(* PLC project multi-phase-flow-facility, Generated TextualNotationConverter 1.0 *)
(* stored: creationDateTime 2025-07-30T12:00:00, modificationDateTime 2025-01-30T12:00:00 *)

FUNCTION_BLOCK ANALOG_IN
  VAR_INPUT
    Name : STRING;
    Description : STRING;
    Raw_Signal : REAL;
    PV_High : REAL;
    PV_Low : REAL;
    Scaling_Slope : REAL;
    Scaling_Offset : REAL;
    Alarm_Enable : BOOL;
  END_VAR
  VAR_OUTPUT
    PV : REAL;
    High_Alarm : BOOL;
    Low_Alarm : BOOL;
    General_Fault : BOOL;
  END_VAR

            
          
END_FUNCTION_BLOCK

FUNCTION_BLOCK PID_BASIC
  VAR_INPUT
    Name : STRING;
    Description : STRING;
    AUTO : BOOL;
    PV : REAL;
    SP : REAL;
    MV_MIN : REAL;
    MV_MAX : REAL;
    X0 : REAL;
    KP : REAL;
    TR : REAL;
    TD : REAL;
    PV_High : REAL;
    PV_Low : REAL;
    Deviation_Limit : REAL;
    Inhibit : BOOL;
  END_VAR
  VAR_OUTPUT
    PV_High_Alarm : BOOL;
    PV_Low_Alarm : BOOL;
    Deviation_Alarm : BOOL;
    XOUT : REAL;
  END_VAR

            
          
END_FUNCTION_BLOCK

FUNCTION_BLOCK RATIO_CONTROL
  VAR_INPUT
    Name : STRING;
    Description : STRING;
    Auto : BOOL;
    PrimaryPV : REAL;
    SecondaryPV : REAL;
    RatioSP : REAL;
    Bias : REAL;
    TrimKp : REAL;
    TrimTi : STRING;
    MV_MIN : REAL;
    MV_MAX : REAL;
    ManOut : REAL;
    Inhibit : BOOL;
  END_VAR
  VAR_OUTPUT
    SlaveSP : REAL;
    ActiveRatio : REAL;
    RatioErr : REAL;
  END_VAR

            
          
END_FUNCTION_BLOCK

FUNCTION_BLOCK VALVE_ELECTRIC
  VAR_INPUT
    Name : STRING;
    Description : STRING;
    Control_Signal : REAL;
    Manual_Mode : BOOL;
    Manual_Position : REAL;
    Open_Limit : REAL;
    Close_Limit : REAL;
    Timeout : STRING;
    Inhibit : BOOL;
  END_VAR
  VAR_OUTPUT
    Valve_Position : REAL;
    Feedback_Pos : REAL;
    Valve_Moving : BOOL;
    Position_Error : BOOL;
    Alarm : BOOL;
  END_VAR

            
          
END_FUNCTION_BLOCK

PROGRAM Section2
  VAR
    FT404_GasFlow_PV : REAL;
    FT406_LiquidFlow_PV : REAL;
    FFIC402_LiquidFlow_SP : REAL;
    FIC406_MV_ToCV406 : REAL;
    PT403_SeparatorPressure_PV : REAL;
    PT408_AuxPressure_PV : REAL;
    PIC401_MV_ToCV401 : REAL;
  END_VAR
  VAR
    FT-404 : ANALOG_IN;
    FT-406 : ANALOG_IN;
    PT-403 : ANALOG_IN;
    PT-408 : ANALOG_IN;
    FFIC-402 : RATIO_CONTROL;
    FIC-406 : PID_BASIC;
    CV-406 : VALVE_ELECTRIC;
    PIC-401 : PID_BASIC;
    CV-401 : VALVE_ELECTRIC;
  END_VAR
  VAR  (* added by the conversion: wires and edge detectors of the diagram *)
    _OR1_OUT : BOOL;
  END_VAR

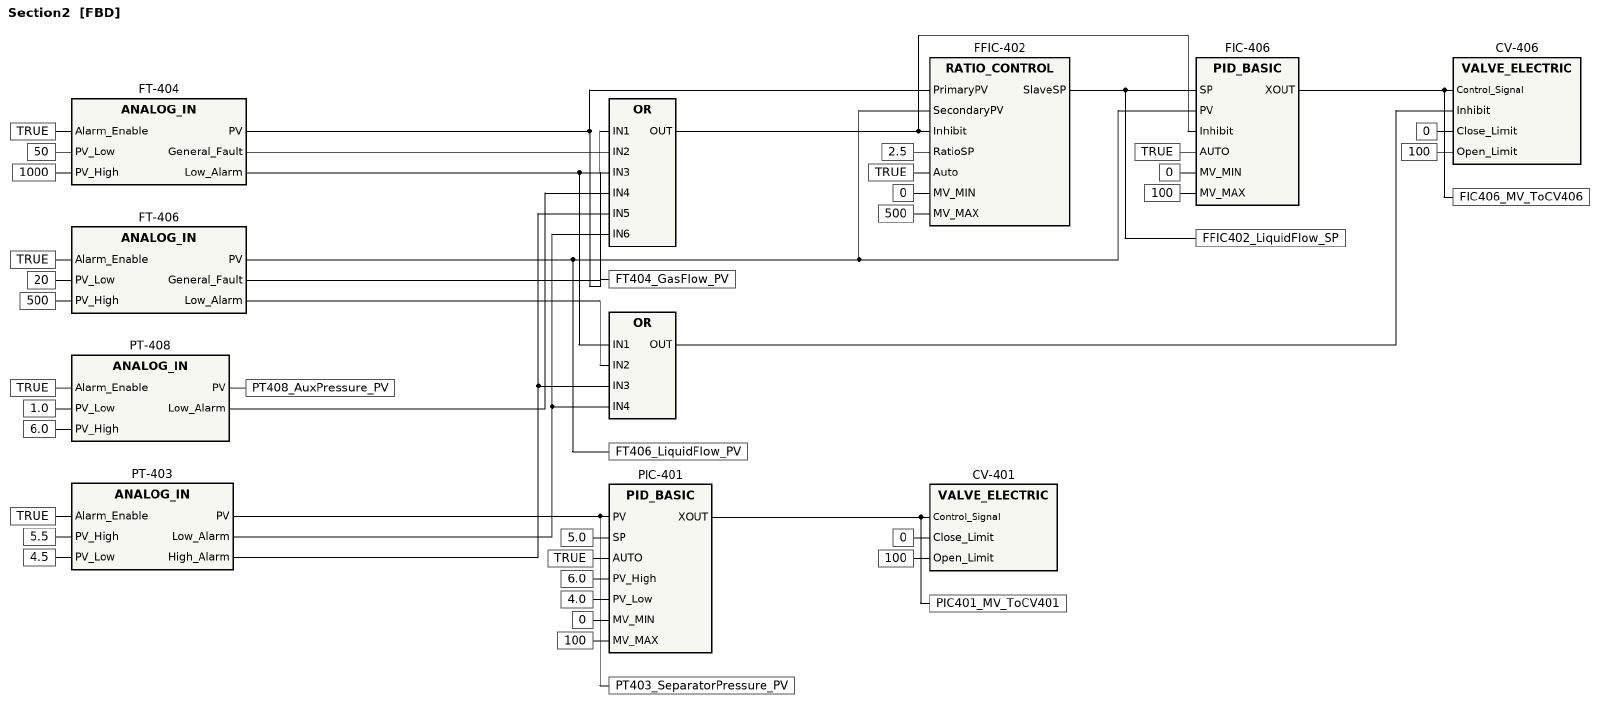
(* FBD diagram, written out as Structured Text *)
FT-404(Alarm_Enable := TRUE, PV_Low := 50, PV_High := 1000);
FT-406(Alarm_Enable := TRUE, PV_Low := 20, PV_High := 500);
PT-408(Alarm_Enable := TRUE, PV_Low := 1.0, PV_High := 6.0);
PT-403(Alarm_Enable := TRUE, PV_High := 5.5, PV_Low := 4.5);
_OR1_OUT := FT-404.Low_Alarm OR FT-404.General_Fault OR FT-406.General_Fault OR PT-408.Low_Alarm OR PT-403.High_Alarm OR PT-403.Low_Alarm;
FFIC-402(PrimaryPV := FT-404.PV, SecondaryPV := FT-406.PV, Inhibit := _OR1_OUT, RatioSP := 2.5, Auto := TRUE, MV_MIN := 0, MV_MAX := 500);
FFIC402_LiquidFlow_SP := FFIC-402.SlaveSP;
FIC-406(SP := FFIC-402.SlaveSP, PV := FT-406.PV, Inhibit := _OR1_OUT, AUTO := TRUE, MV_MIN := 0, MV_MAX := 100);
FIC406_MV_ToCV406 := FIC-406.XOUT;
FT404_GasFlow_PV := FT-404.PV;
FT406_LiquidFlow_PV := FT-406.PV;
PIC-401(PV := PT-403.PV, SP := 5.0, AUTO := TRUE, PV_High := 6.0, PV_Low := 4.0, MV_MIN := 0, MV_MAX := 100);
PIC401_MV_ToCV401 := PIC-401.XOUT;
PT403_SeparatorPressure_PV := PT-403.PV;
PT408_AuxPressure_PV := PT-408.PV;
CV-406(Control_Signal := FIC-406.XOUT, Inhibit := FT-404.Low_Alarm OR FT-406.Low_Alarm OR PT-403.High_Alarm OR PT-403.Low_Alarm, Close_Limit := 0, Open_Limit := 100);
CV-401(Control_Signal := PIC-401.XOUT, Close_Limit := 0, Open_Limit := 100);
END_PROGRAM

FUNCTION_BLOCK BOOL_IN
  VAR_INPUT
    Name : STRING;
    Description : STRING;
    Bool_In : BOOL;
    Alarm_OnTrue : BOOL;
    Alarm_OnFalse : BOOL;
    Latch_Enable : BOOL;
    Reset_Latch : BOOL;
  END_VAR
  VAR_OUTPUT
    Bool_Out : BOOL;
    Alarm_Active : BOOL;
    Latched_Status : BOOL;
  END_VAR

            
          
END_FUNCTION_BLOCK

FUNCTION_BLOCK DIGITAL_IN
  VAR_INPUT
    Name : STRING;
    Description : STRING;
    DI_Raw : BOOL;
    DebounceTime : STRING;
    EnableAlarm : BOOL;
  END_VAR
  VAR_OUTPUT
    DI_Out : BOOL;
    Fault_State : BOOL;
  END_VAR

            
          
END_FUNCTION_BLOCK

FUNCTION_BLOCK DUTY_STANDBY
  VAR_INPUT
    Name : STRING;
    Description : STRING;
    Enable : BOOL;
    StartRequest : BOOL;
    AlternateEnable : BOOL;
    ForcePumpA : BOOL;
    ForcePumpB : BOOL;
    DutyElapsed : BOOL;
    MinRunElapsed : BOOL;
    SwitchoverDelayElapsed : BOOL;
    StartTimeoutElapsed : BOOL;
    PumpA_RunFB : BOOL;
    PumpB_RunFB : BOOL;
    PumpA_Fault : BOOL;
    PumpB_Fault : BOOL;
    Reset : BOOL;
    Inhibit : BOOL;
  END_VAR
  VAR_OUTPUT
    CmdPumpA : BOOL;
    CmdPumpB : BOOL;
    ActiveIsA : BOOL;
    SwitchedDueToDuty : BOOL;
    SwitchedDueToFailure : BOOL;
    Alarm_FailedStart_A : BOOL;
    Alarm_FailedStart_B : BOOL;
    Alarm_NoAvailablePump : BOOL;
  END_VAR

            
          
END_FUNCTION_BLOCK

FUNCTION_BLOCK MOTOR_2SPD
  VAR_INPUT
    Name : STRING;
    Description : STRING;
    Start_Cmd : BOOL;
    Stop_Cmd : BOOL;
    Speed_High_Cmd : BOOL;
    Speed_Low_Cmd : BOOL;
    Inhibit : BOOL;
  END_VAR
  VAR_OUTPUT
    Motor_Start_Out : BOOL;
    FB_Running : BOOL;
    FB_Trip : BOOL;
    FB_HighSpeed : BOOL;
    FB_LowSpeed : BOOL;
    Alarm_Speed_Error : BOOL;
  END_VAR

            
          
END_FUNCTION_BLOCK

FUNCTION_BLOCK MOTOR_ON_OFF
  VAR_INPUT
    Name : STRING;
    Description : STRING;
    Start_Cmd : BOOL;
    Stop_Cmd : BOOL;
    Start_Delay : STRING;
    MinRunTime : STRING;
    Inhibit : BOOL;
  END_VAR
  VAR_OUTPUT
    Motor_Start_Out : BOOL;
    FB_Running : BOOL;
    FB_Trip : BOOL;
    Alarm_Start_Fail : BOOL;
    Alarm_Stop_Fail : BOOL;
  END_VAR

            
          
END_FUNCTION_BLOCK

FUNCTION_BLOCK MOTOR_VSD
  VAR_INPUT
    Name : STRING;
    Description : STRING;
    Start_Cmd : BOOL;
    Stop_Cmd : BOOL;
    Speed_SP : REAL;
    Accel_Ramp : STRING;
    Decel_Ramp : STRING;
    Inhibit : BOOL;
  END_VAR
  VAR_OUTPUT
    Speed_Out : REAL;
    FB_Running : BOOL;
    FB_Fault : BOOL;
    FB_Ready : BOOL;
    FB_ActualSpeed : REAL;
    Alarm_Speed_Deviation : BOOL;
    Alarm_Comm_Fail : BOOL;
  END_VAR

            
          
END_FUNCTION_BLOCK

FUNCTION_BLOCK SPLIT_RANGE
  VAR_INPUT
    Name : STRING;
    Description : STRING;
    IN : REAL;
    Split_Point : REAL;
    Output1_Start : REAL;
    Output1_End : REAL;
    Output2_Start : REAL;
    Output2_End : REAL;
  END_VAR
  VAR_OUTPUT
    OUT1 : REAL;
    OUT2 : REAL;
  END_VAR

            
          
END_FUNCTION_BLOCK

FUNCTION_BLOCK VALVE_ON_OFF
  VAR_INPUT
    Name : STRING;
    Description : STRING;
    Open_Cmd : BOOL;
    Close_Cmd : BOOL;
    Timeout : STRING;
    Inhibit : BOOL;
  END_VAR
  VAR_OUTPUT
    FB_Opened : BOOL;
    FB_Closed : BOOL;
    Valve_Open_Out : BOOL;
    Valve_Close_Out : BOOL;
    Alarm_Position_Error : BOOL;
    Alarm_General : BOOL;
  END_VAR

            
          
END_FUNCTION_BLOCK

FUNCTION_BLOCK VOTING_ANALOG
  VAR_INPUT
    Name : STRING;
    Description : STRING;
    Input1 : REAL;
    Input2 : REAL;
    Input3 : REAL;
    Deviation_Limit : REAL;
    Voting_Scheme : STRING;
    EnableAlarm : BOOL;
    Inhibit : BOOL;
  END_VAR
  VAR_OUTPUT
    Voted_Output : REAL;
    Sensor1_Fault : BOOL;
    Sensor2_Fault : BOOL;
    Sensor3_Fault : BOOL;
    Alarm_Voting_Error : BOOL;
    Healthy_Sensors_Count : INT;
  END_VAR

            
          
END_FUNCTION_BLOCK

PROGRAM Section3
  VAR
    PT501_PressurePV : REAL;
    LI502_LevelPV : REAL;
    PIC501_ControlOutput : REAL;
  END_VAR
  VAR
    FV-102 : VALVE_ELECTRIC;
    PT-501 : ANALOG_IN;
    LI-502 : ANALOG_IN;
    PIC-501 : PID_BASIC;
  END_VAR

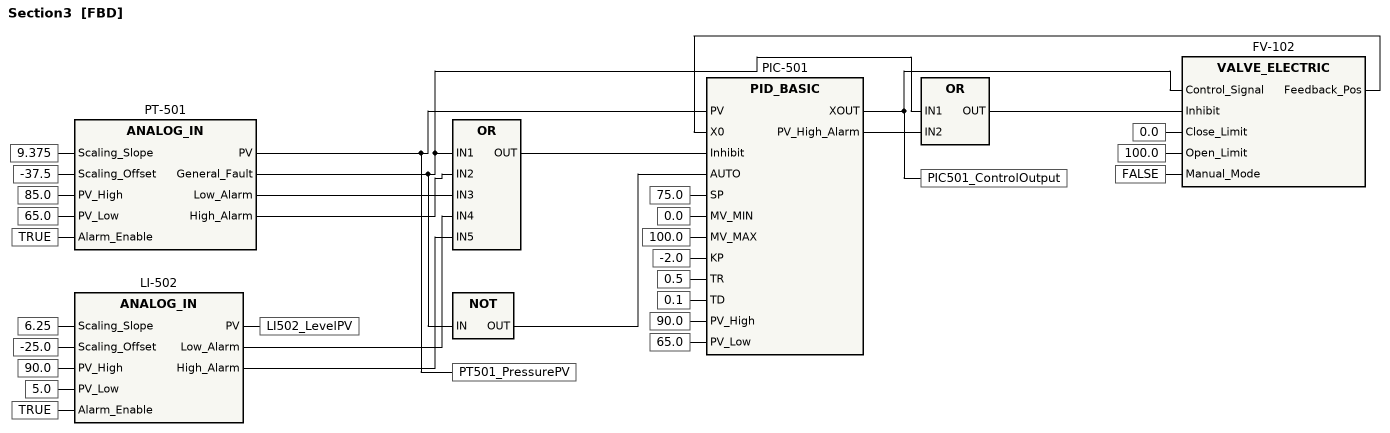
(* FBD diagram, written out as Structured Text *)
LI-502(Scaling_Slope := 6.25, Scaling_Offset := -25.0, PV_High := 90.0, PV_Low := 5.0, Alarm_Enable := TRUE);
LI502_LevelPV := LI-502.PV;
PT-501(Scaling_Slope := 9.375, Scaling_Offset := -37.5, PV_High := 85.0, PV_Low := 65.0, Alarm_Enable := TRUE);
FV-102(Control_Signal := PIC-501.XOUT, Inhibit := PT-501.General_Fault OR PIC-501.PV_High_Alarm, Close_Limit := 0.0, Open_Limit := 100.0, Manual_Mode := FALSE);
PIC-501(PV := PT-501.PV, X0 := FV-102.Feedback_Pos, Inhibit := PT-501.General_Fault OR PT-501.High_Alarm OR PT-501.Low_Alarm OR LI-502.Low_Alarm OR LI-502.High_Alarm, AUTO := NOT PT-501.General_Fault, SP := 75.0, MV_MIN := 0.0, MV_MAX := 100.0, KP := -2.0, TR := 0.5, TD := 0.1, PV_High := 90.0, PV_Low := 65.0);
PIC501_ControlOutput := PIC-501.XOUT;
PT501_PressurePV := PT-501.PV;
END_PROGRAM

PROGRAM Section4
  VAR
    LI201_Level_Pct : REAL;
    FIC302_MV_Percent_To_FV101 : REAL;
    FV101_Feedback_Position_Pct : REAL;
    XV010_Open_Feedback : BOOL;
    XV011_Open_Feedback : BOOL;
  END_VAR
  VAR
    FIC-302 : PID_BASIC;
    FV-101 : VALVE_ELECTRIC;
    LI-201 : ANALOG_IN;
    XV-010 : VALVE_ON_OFF;
    XV-011 : VALVE_ON_OFF;
  END_VAR
  VAR  (* added by the conversion: wires and edge detectors of the diagram *)
    _OR81_OUT : BOOL;
    _OR82_OUT : BOOL;
  END_VAR

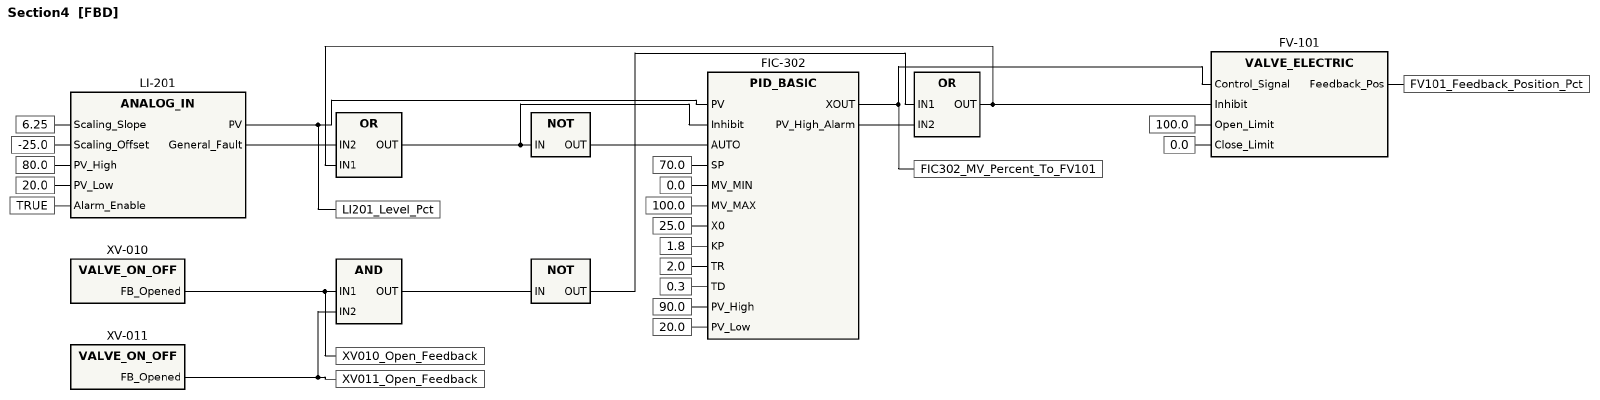
(* FBD diagram, written out as Structured Text *)
LI-201(Scaling_Slope := 6.25, Scaling_Offset := -25.0, PV_High := 80.0, PV_Low := 20.0, Alarm_Enable := TRUE);
XV-010();
XV-011();
_OR81_OUT := NOT (XV-010.FB_Opened AND XV-011.FB_Opened) OR FIC-302.PV_High_Alarm;
_OR82_OUT := LI-201.General_Fault OR _OR81_OUT;
FIC-302(PV := LI-201.PV, Inhibit := _OR82_OUT, AUTO := NOT _OR82_OUT, SP := 70.0, MV_MIN := 0.0, MV_MAX := 100.0, X0 := 25.0, KP := 1.8, TR := 2.0, TD := 0.3, PV_High := 90.0, PV_Low := 20.0);
FIC302_MV_Percent_To_FV101 := FIC-302.XOUT;
FV-101(Control_Signal := FIC-302.XOUT, Inhibit := _OR81_OUT, Open_Limit := 100.0, Close_Limit := 0.0);
FV101_Feedback_Position_Pct := FV-101.Feedback_Pos;
LI201_Level_Pct := LI-201.PV;
XV010_Open_Feedback := XV-010.FB_Opened;
XV011_Open_Feedback := XV-011.FB_Opened;
END_PROGRAM

PROGRAM Section5
  VAR
    FV103_ControlSignal_From_FIC101 : REAL;
    P001_SpeedCmd_From_FIC102 : REAL;
    LevelTrip : BOOL;
    PumpStartPermissive : BOOL;
    ValveOpenPermit : BOOL;
    FT102_FlowAbove10 : BOOL;
    FlowValid_DelayOK : BOOL;
    ValveOpenFB_OK : BOOL;
    FIC101_DeviationAlarm_15s : BOOL;
    FIC102_DeviationAlarm_15s : BOOL;
  END_VAR
  VAR
    FT-102 : ANALOG_IN;
    FT-104 : ANALOG_IN;
    LI-101 : ANALOG_IN;
    FIC-101 : PID_BASIC;
    FIC-102 : PID_BASIC;
    FV-103 : VALVE_ELECTRIC;
    P-001 : MOTOR_VSD;
    FT102_Flow_Valid_TON : TON;
    FIC101_DevAlarm_TON : TON;
    FIC102_DevAlarm_TON : TON;
  END_VAR
  VAR  (* added by the conversion: wires and edge detectors of the diagram *)
    _NOT111_OUT : BOOL;
    _AND121_OUT : BOOL;
  END_VAR

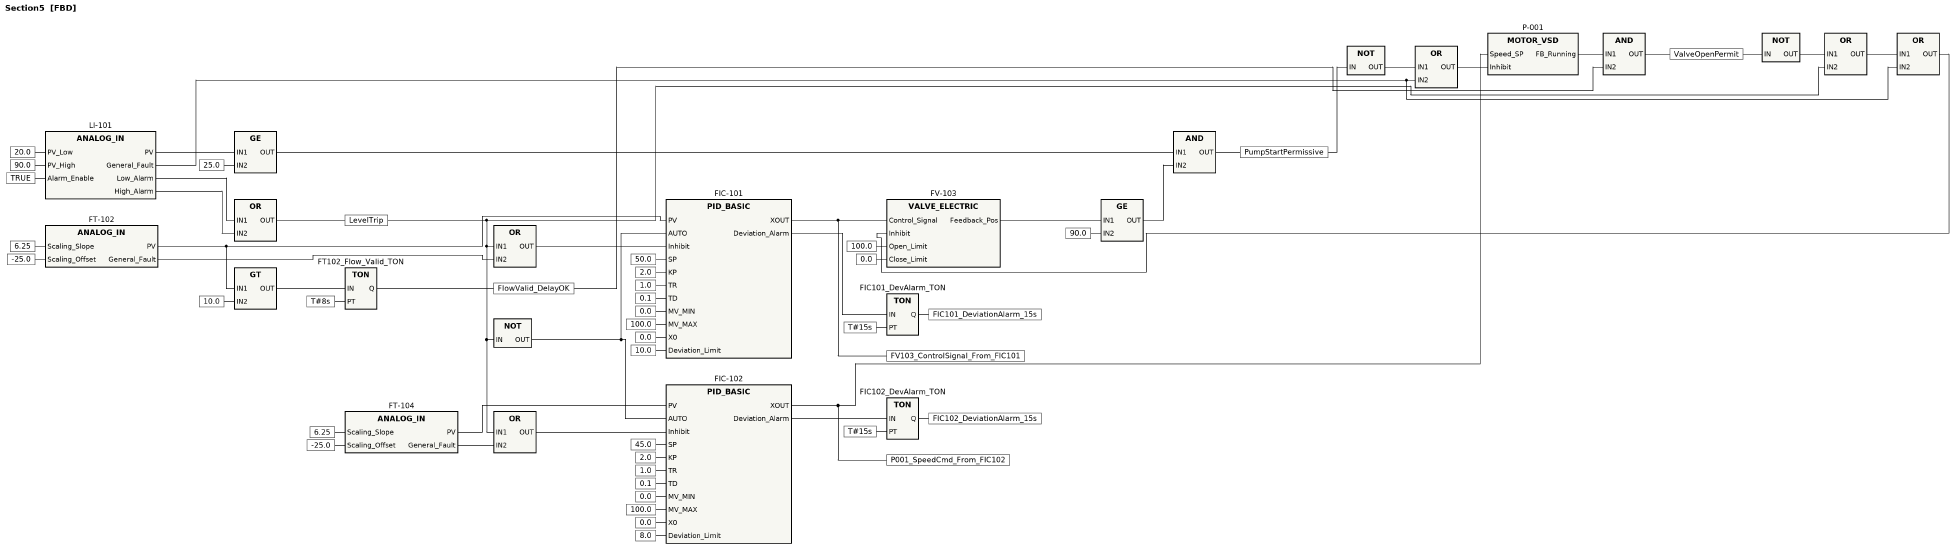
(* FBD diagram, written out as Structured Text *)
FT-102(Scaling_Slope := 6.25, Scaling_Offset := -25.0);
LI-101(PV_Low := 20.0, PV_High := 90.0, Alarm_Enable := TRUE);
_NOT111_OUT := NOT (LI-101.Low_Alarm OR LI-101.High_Alarm);
FIC-101(PV := FT-102.PV, AUTO := _NOT111_OUT, Inhibit := LI-101.Low_Alarm OR LI-101.High_Alarm OR FT-102.General_Fault, SP := 50.0, KP := 2.0, TR := 1.0, TD := 0.1, MV_MIN := 0.0, MV_MAX := 100.0, X0 := 0.0, Deviation_Limit := 10.0);
FIC101_DevAlarm_TON(IN := FIC-101.Deviation_Alarm, PT := T#15s);
FIC101_DeviationAlarm_15s := FIC101_DevAlarm_TON.Q;
FT-104(Scaling_Slope := 6.25, Scaling_Offset := -25.0);
FIC-102(PV := FT-104.PV, AUTO := _NOT111_OUT, Inhibit := LI-101.Low_Alarm OR LI-101.High_Alarm OR FT-104.General_Fault, SP := 45.0, KP := 2.0, TR := 1.0, TD := 0.1, MV_MIN := 0.0, MV_MAX := 100.0, X0 := 0.0, Deviation_Limit := 8.0);
FIC102_DevAlarm_TON(IN := FIC-102.Deviation_Alarm, PT := T#15s);
FIC102_DeviationAlarm_15s := FIC102_DevAlarm_TON.Q;
FV103_ControlSignal_From_FIC101 := FIC-101.XOUT;
FT102_Flow_Valid_TON(IN := FT-102.PV > 10.0, PT := T#8s);
FlowValid_DelayOK := FT102_Flow_Valid_TON.Q;
LevelTrip := LI-101.Low_Alarm OR LI-101.High_Alarm;
P001_SpeedCmd_From_FIC102 := FIC-102.XOUT;
P-001(Speed_SP := FIC-102.XOUT, Inhibit := NOT _AND121_OUT OR LI-101.General_Fault);
FV-103(Control_Signal := FIC-101.XOUT, Inhibit := NOT (P-001.FB_Running AND FT102_Flow_Valid_TON.Q) OR LI-101.Low_Alarm OR LI-101.High_Alarm OR LI-101.General_Fault, Open_Limit := 100.0, Close_Limit := 0.0);
_AND121_OUT := LI-101.PV >= 25.0 AND FV-103.Feedback_Pos >= 90.0;
PumpStartPermissive := _AND121_OUT;
ValveOpenPermit := P-001.FB_Running AND FT102_Flow_Valid_TON.Q;
END_PROGRAM

PROGRAM Section6
  VAR
    FT105_FlowRate_PV : REAL;
    LI503_Level_PV : REAL;
    LIC502_XOUT_to_LVC502 : REAL;
    LIC503_XOUT_to_LVC507 : REAL;
  END_VAR
  VAR
    FT-105 : ANALOG_IN;
    LI-503 : ANALOG_IN;
    LIC-502 : PID_BASIC;
    LIC-503 : PID_BASIC;
    LVC-502 : VALVE_ELECTRIC;
    LVC-507 : VALVE_ELECTRIC;
    P-001 : MOTOR_ON_OFF;
  END_VAR
  VAR  (* added by the conversion: wires and edge detectors of the diagram *)
    _NOT173_OUT : MOTOR_ON_OFF;
    _OR174_OUT : ANALOG_IN;
    _OR175_OUT : ANALOG_IN;
  END_VAR

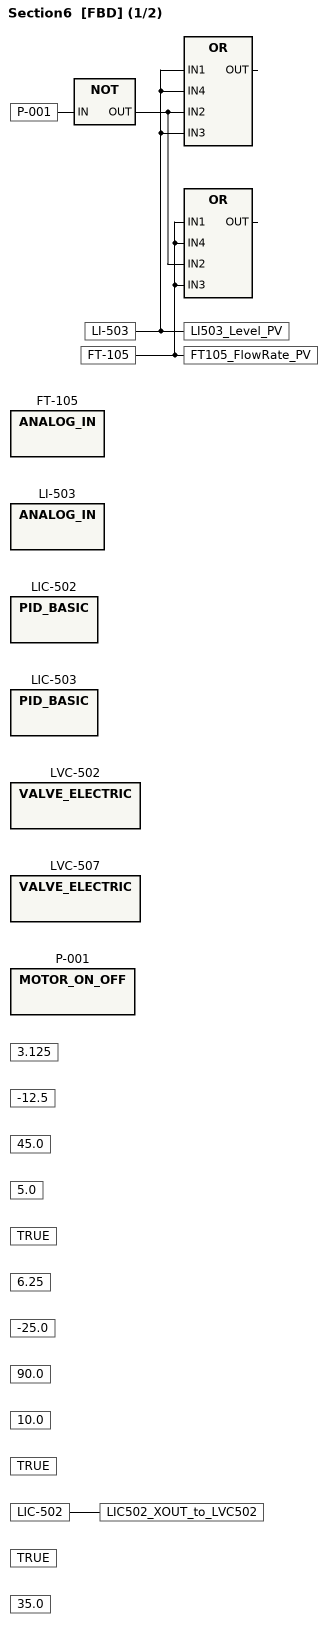
(* FBD diagram, written out as Structured Text *)
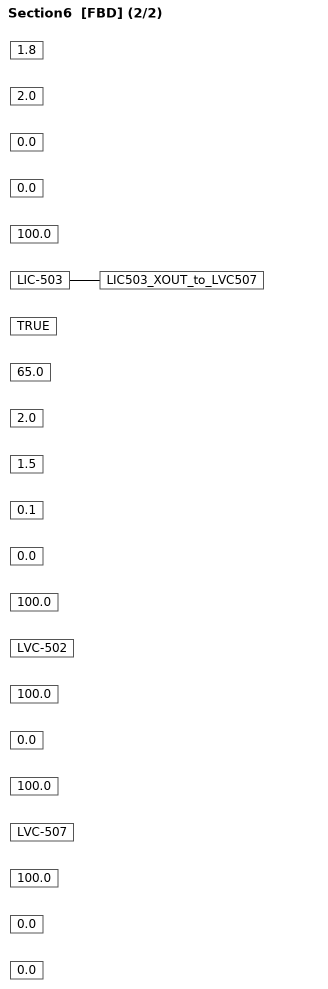
FT105_FlowRate_PV := FT-105;
LI503_Level_PV := LI-503;
LIC502_XOUT_to_LVC502 := LIC-502;
LIC503_XOUT_to_LVC507 := LIC-503;
_NOT173_OUT := NOT (P-001);
_OR174_OUT := (LI-503) OR (LI-503) OR _NOT173_OUT OR (LI-503);
_OR175_OUT := (FT-105) OR (FT-105) OR _NOT173_OUT OR (FT-105);
FT-105();
LI-503();
LIC-502();
LIC-503();
LVC-502();
LVC-507();
P-001();
(* drawn but not wired to any output: 3.125, -12.5, 45.0, 5.0, TRUE, 6.25, -25.0, 90.0, 10.0, TRUE, TRUE, 35.0, 1.8, 2.0, 0.0, 0.0, 100.0, TRUE, 65.0, 2.0, 1.5, 0.1, 0.0, 100.0, LVC-502, 100.0, 0.0, 100.0, LVC-507, 100.0, 0.0, 0.0 *)
END_PROGRAM

PROGRAM Section7
  VAR
    PIT106_PressurePV : REAL;
    PIC105_MV_Output : REAL;
  END_VAR
  VAR
    PIT-106 : ANALOG_IN;
    PIC-105 : PID_BASIC;
    V-010 : VALVE_ELECTRIC;
    COMPRESSOR_RUN_PERMISSIVE : BOOL_IN;
    StartupDelay_TON : TON;
  END_VAR
  VAR  (* added by the conversion: wires and edge detectors of the diagram *)
    _OR225_OUT : BOOL_IN;
  END_VAR

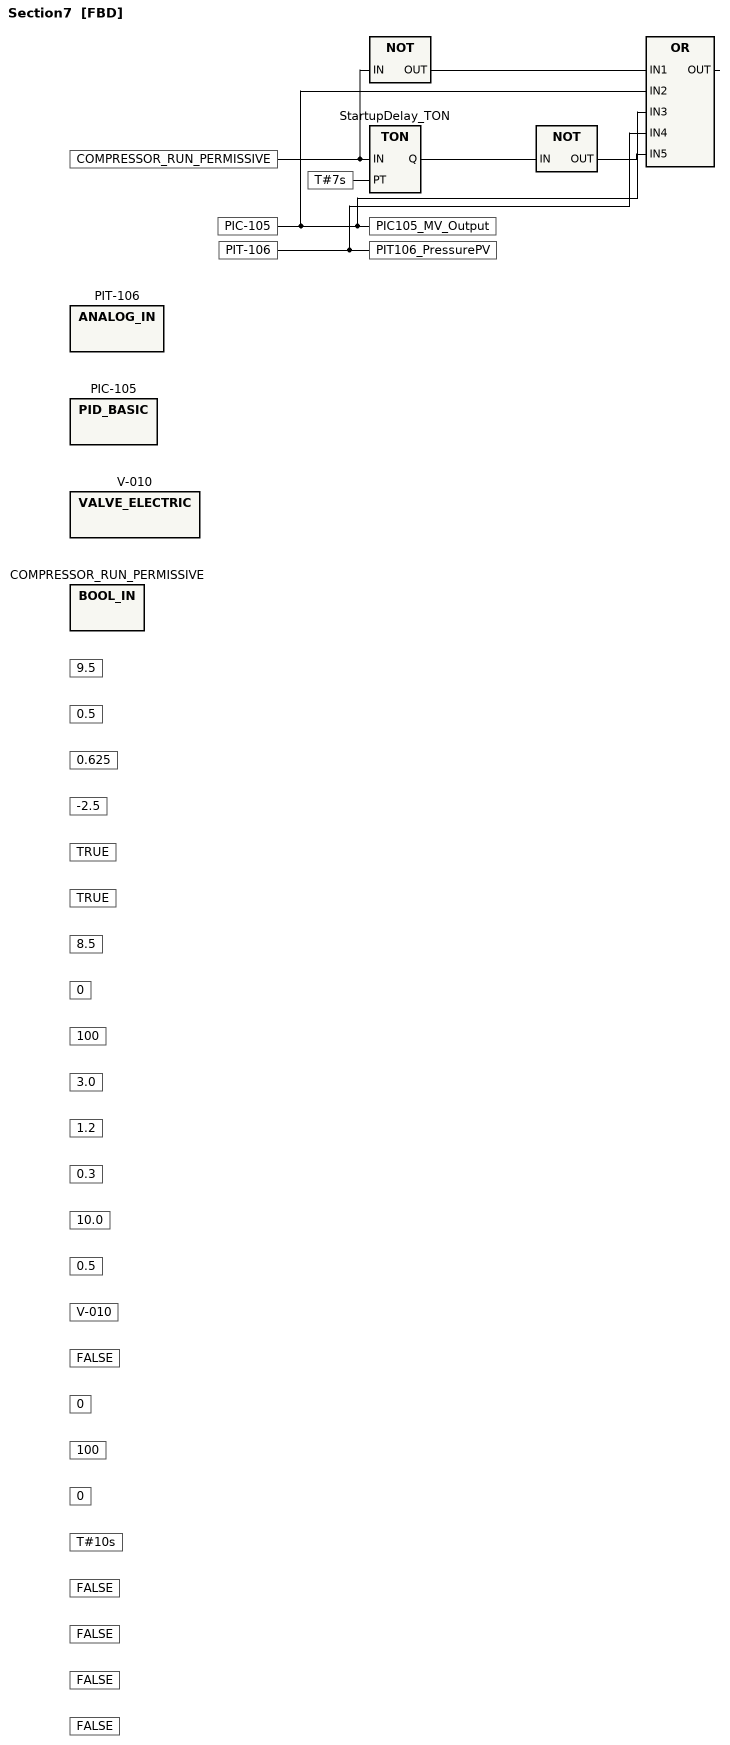
(* FBD diagram, written out as Structured Text *)
PIC105_MV_Output := PIC-105;
PIT106_PressurePV := PIT-106;
StartupDelay_TON(IN := COMPRESSOR_RUN_PERMISSIVE, PT := T#7s);
_OR225_OUT := NOT COMPRESSOR_RUN_PERMISSIVE OR (PIC-105) OR (PIC-105) OR (PIT-106) OR NOT StartupDelay_TON.Q;
PIT-106();
PIC-105();
V-010();
COMPRESSOR_RUN_PERMISSIVE();
(* drawn but not wired to any output: 9.5, 0.5, 0.625, -2.5, TRUE, TRUE, 8.5, 0, 100, 3.0, 1.2, 0.3, 10.0, 0.5, V-010, FALSE, 0, 100, 0, T#10s, FALSE, FALSE, FALSE, FALSE *)
END_PROGRAM

CONFIGURATION Config0
  RESOURCE Res0 ON PLC
    TASK task0(INTERVAL := T#20ms, PRIORITY := 0);
    PROGRAM instance0 WITH task0 : Section2;
    PROGRAM instance_1 WITH task0 : Section3;
    PROGRAM instance_2 WITH task0 : Section4;
    PROGRAM instance_3 WITH task0 : Section5;
    PROGRAM instance_4 WITH task0 : Section6;
    PROGRAM instance_5 WITH task0 : Section7;
  END_RESOURCE
END_CONFIGURATION
